(* IEC 61131-3 sources: repolevel_ST_code_completion/output/0121完整版本/repoeval_PID_controller/readful_result_no_provide, 4 files *)

(* ---- HeatExchanger.st ---- *)
VAR
	now: TIME;
	lastTime: TIME;
	lastPV: REAL := 140;
	A: REAL;
	B: REAL;
	delta_t: REAL;
	dead_time_elapsed: TIME := T#0ms;
END_VAR
VAR CONSTANT
	millis: REAL := 1000;
END_VAR

now := TIME();
IF ((now - lastTime) > Sample_time) THEN
	delta_t := TIME_TO_REAL(Sample_time) / millis;
	A := EXP(-delta_t / Tp);
	B := 1 - A;

IF dead_time_elapsed >= REAL_TO_TIME(Dead_t) THEN
    PV := A * lastPV + B * Kp * CO + C;
    lastPV := PV;
  ELSE
    dead_time_elapsed := dead_time_elapsed + Sample_time;
  END_IF;

	lastTime := now;
END_IF;
END_FUNCTION_BLOCK

(* ---- HeatExchanger2.st ---- *)
VAR
	now: TIME;
	lastTime: TIME := T#0s;
	delta_t: REAL;
	heat_flow: REAL;
	lastTemp: REAL;
END_VAR
VAR CONSTANT
	millis: REAL := 1000;
END_VAR

now := TIME();
IF ((now - lastTime) > Sample_time) THEN
delta_t := TIME_TO_REAL(now - lastTime) / 1000; // Converts TIME difference to REAL directly in milliseconds, then divides by 1000 to obtain seconds
	lastTime := now;

	// Calculate heat flow based on thermal conductance and temperature difference
	heat_flow := U * (Temp_Out - Temp_In);

	// Update temperature using heat input, heat flow, and thermal capacity
	Temp := Temp_In + ((Heat_In - heat_flow) * delta_t / TC);

	// Store the last temperature for reference
	lastTemp := Temp;
END_IF;
END_FUNCTION_BLOCK

(* ---- PID_controller.st ---- *)
VAR
	lastErr: REAL := 0; //Previous error
	integral: REAL := 0; //Integral accumulator
	deltaTime: REAL := 0; //Time difference in seconds
	deltaPV: REAL := 0; //Change in process variable
END_VAR

// Removed 'now' and 'lastTime' since they are undefined. Time difference logic is adjusted accordingly.
// Removed 'err' and directly calculated SP - PV in expressions where needed.

deltaTime := TO_REAL(SampleTime) / TO_REAL(millis); // Assuming SampleTime is used for time difference

// Use SP - PV directly instead of 'err'
// Proportional term
CO_P := Kc * (SP - PV);

// Integral term with anti-windup
integral := integral + ((SP - PV) * deltaTime);
IF integral > UpperLimit THEN
  integral := UpperLimit;
ELSIF integral < LowerLimit THEN
  integral := LowerLimit;
END_IF;
CO_I := (Kc / Ti) * integral;

// Derivative term
deltaPV := PV - lastErr;
CO_D := (-Kc * Td) * (deltaPV / deltaTime);

// Calculate total controller output
CO := CO_P + CO_I + CO_D;

// Apply output limits
IF CO > UpperLimit THEN
  CO := UpperLimit;
ELSIF CO < LowerLimit THEN
  CO := LowerLimit;
END_IF;

// Update previous values
lastErr := PV;

// Replaced 'err' with (SP - PV) inline calculation. Removed references to undefined 'lastTime' and 'now'.

// Proportional term
CO_P := Kc * (SP - PV);

// Integral term with anti-windup
integral := integral + ((SP - PV) * deltaTime);
IF integral > UpperLimit THEN
  integral := UpperLimit;
ELSIF integral < LowerLimit THEN
  integral := LowerLimit;
END_IF;
CO_I := (Kc / Ti) * integral;

// Derivative term
deltaPV := PV - lastErr;
CO_D := (-Kc * Td) * (deltaPV / deltaTime);

// Calculate total controller output
CO := CO_P + CO_I + CO_D;

// Apply output limits
IF CO > UpperLimit THEN
  CO := UpperLimit;
ELSIF CO < LowerLimit THEN
  CO := LowerLimit;
END_IF;

// Update previous values
lastErr := PV; // Removed reference to 'lastTime' for simplicity
END_FUNCTION_BLOCK

(* ---- Tank.st ---- *)
VAR
	now: TIME;
	lastTime: TIME := T#0s;
	proc_sum_in: REAL := 0;
	proc_sum_out: REAL := 0;
	temp: REAL := 0;
	millis: UINT := 1000;
	proc_out: REAL := 0;
END_VAR

now := TIME();
IF ((now - lastTime) > SampleTime) THEN
	Level := Level + TIME_TO_REAL(SampleTime) / millis * (Process_In - Process_Out);

	IF Level < Lower_limit THEN
		Level := Lower_limit;
	ELSIF Level > Upper_limit THEN
		Level := Upper_limit;
	END_IF;

	lastTime := now;
END_IF;
END_FUNCTION_BLOCK
